// TIA Portal V19 export
FUNCTION_BLOCK "TYPIC_C104_IF_NSA"   // FB92, FBD
TITLE = TYPIC_C104_IF_NSA: Noodstroomaggregaat
{ S7_Optimized_Access := 'TRUE' }
AUTHOR : OCOTECH
FAMILY : Typical
NAME : C104.702
// Logisch Object Besturing: C104.702
// 
// De interne functie Noodstroomaggregaat verzorgt de bewaking van een noodstroomaggregaat.
// stored: MemoryReserve 10, SetENOAutomatically false
   VAR_INPUT
      EXT_AUT { ExternalAccessible := 'False'; ExternalVisible := 'False'; ExternalWritable := 'False'} : Bool;   // Externe (hoofd) beveiliging (1 = OK)
      EXT_HW { ExternalAccessible := 'False'; ExternalVisible := 'False'; ExternalWritable := 'False'} : Bool;   // Sturings hardware (PLC) bewaking (1 = OK)
      IN_STO_NOK { ExternalAccessible := 'False'; ExternalVisible := 'False'; ExternalWritable := 'False'} : Bool;   // Storing aanwezig die niet observeerbaar tot gevolg heeft
      IN_STO_OK { ExternalAccessible := 'False'; ExternalVisible := 'False'; ExternalWritable := 'False'} : Bool;   // Storing aanwezig die observeerbaarheid niet beinvloed
      IN_ENE { ExternalAccessible := 'False'; ExternalVisible := 'False'; ExternalWritable := 'False'} : Real;   // Geleverde energie per aggregaat
      IN_PHI { ExternalAccessible := 'False'; ExternalVisible := 'False'; ExternalWritable := 'False'} : Real;   // Fasehoek (cos phi)
      IN_SPA1 { ExternalAccessible := 'False'; ExternalVisible := 'False'; ExternalWritable := 'False'} : Real;   // Spanningsniveau lijn 1
      IN_SPA2 { ExternalAccessible := 'False'; ExternalVisible := 'False'; ExternalWritable := 'False'} : Real;   // Spanningsniveau lijn 2
      IN_SPA3 { ExternalAccessible := 'False'; ExternalVisible := 'False'; ExternalWritable := 'False'} : Real;   // Spanningsniveau lijn 3
      IN_STR { ExternalAccessible := 'False'; ExternalVisible := 'False'; ExternalWritable := 'False'} : Real;   // Stroomsterkte
      IN_WRE { ExternalAccessible := 'False'; ExternalVisible := 'False'; ExternalWritable := 'False'} : Bool;   // TRUE = werkingsregime: Belast FALSE = werkingsregime: Onbelast
      IN_STS1 { ExternalAccessible := 'False'; ExternalVisible := 'False'; ExternalWritable := 'False'} : Bool;   // Status: Standby
      IN_STS2 { ExternalAccessible := 'False'; ExternalVisible := 'False'; ExternalWritable := 'False'} : Bool;   // Status: Storing
      IN_STS3 { ExternalAccessible := 'False'; ExternalVisible := 'False'; ExternalWritable := 'False'} : Bool;   // Status: Uitgeschakeld
      IN_STS4 { ExternalAccessible := 'False'; ExternalVisible := 'False'; ExternalWritable := 'False'} : Bool;   // Status: Test
      IN_STS_AAN { ExternalAccessible := 'False'; ExternalVisible := 'False'; ExternalWritable := 'False'} : Bool;   // In bedrijf (Aan)
      IN_LDE { ExternalAccessible := 'False'; ExternalVisible := 'False'; ExternalWritable := 'False'} : Bool;   // Lekdetectie NSA
      IN_TYD_TOT_AAN_UUR { ExternalAccessible := 'False'; ExternalVisible := 'False'; ExternalWritable := 'False'} : LInt;   // TYD_TOT_AAN_UUR
      IN_SNS { ExternalAccessible := 'False'; ExternalVisible := 'False'; ExternalWritable := 'False'} : Bool;   // Noodstop (1 = gedeactiveerd)
      IN_OPT_LDE { ExternalAccessible := 'False'; ExternalVisible := 'False'; ExternalWritable := 'False'} : Bool;   // Lekdetectie brandstof dagtank
      IN_OPT_NIV { ExternalAccessible := 'False'; ExternalVisible := 'False'; ExternalWritable := 'False'} : Real;   // Brandstof niveau brandstof dagtank
      IN_OPT_HOOG { ExternalAccessible := 'False'; ExternalVisible := 'False'; ExternalWritable := 'False'} : Bool;   // Overvulbeveiliging brandstof dagtank aangesproken
      IN_OPT_STO { ExternalAccessible := 'False'; ExternalVisible := 'False'; ExternalWritable := 'False'} : Bool;   // Dagtank noodstroomaggregaat in storing
      IN_AUT_C104 { ExternalAccessible := 'False'; ExternalVisible := 'False'; ExternalWritable := 'False'} : Bool;   // Beveiligingen: serie geschakelde terugmelding (1 = OK)
   END_VAR
   VAR_OUTPUT
      VAR_IF_NSA { ExternalAccessible := 'False'; ExternalVisible := 'False'; ExternalWritable := 'False'} : "C104_VAR_IF_NSA_TYPIC";   // Struct met alle variabelen naar bovenliggende functies
   END_VAR
   VAR
      STO { ExternalWritable := 'False'} : Struct   // Storingen
         A001 : Bool;   // Beveiliging aangesproken
         A002 : Bool;   // Noodstroomaggregaat in storing
         A003 : Bool;   // Algemene storing noodstroomaggregaat
         A004 : Bool;   // Lekdetectie NSA
         A005 : Bool;   // Noodstop van het noodstroomaggregaat is geactiveerd
         A006 : Bool;   // Dagtank noodstroomaggregaat in storing
         A007 : Bool;   // Lekdetectie brandstof dagtank
         A008 : Bool;   // Overvulbeveiliging brandstof dagtank aangesproken
      END_STRUCT;
      VAR { ExternalWritable := 'False'} : Struct   // Variabelen
         ENE { ExternalAccessible := 'False'; ExternalVisible := 'False'} : Real;   // Geleverde energie per aggregaat [kWh]
         PHI { ExternalAccessible := 'False'; ExternalVisible := 'False'} : Real;   // Fasehoek (cos phi)
         SPA1 { ExternalAccessible := 'False'; ExternalVisible := 'False'} : Real;   // Spanningsniveau lijn 1
         SPA2 { ExternalAccessible := 'False'; ExternalVisible := 'False'} : Real;   // Spanningsniveau lijn 2
         SPA3 { ExternalAccessible := 'False'; ExternalVisible := 'False'} : Real;   // Spanningsniveau lijn 3
         STR { ExternalAccessible := 'False'; ExternalVisible := 'False'} : Real;   // Stroomsterkte
         WRE { ExternalAccessible := 'False'; ExternalVisible := 'False'} : Bool;   // TRUE = werkingsregime: Belast FALSE = werkingsregime: Onbelast
         STS1 { ExternalAccessible := 'False'; ExternalVisible := 'False'} : Bool;   // Status: Standby
         STS2 { ExternalAccessible := 'False'; ExternalVisible := 'False'} : Bool;   // Status: Storing
         STS3 { ExternalAccessible := 'False'; ExternalVisible := 'False'} : Bool;   // Status: Uitgeschakeld
         STS4 { ExternalAccessible := 'False'; ExternalVisible := 'False'} : Bool;   // Status: Test
         STS_AAN { ExternalAccessible := 'False'; ExternalVisible := 'False'} : Bool;   // In bedrijf (AAN)
         LDE { ExternalAccessible := 'False'; ExternalVisible := 'False'} : Bool;   // Lekdetectie NSA
         TYD_TOT_AAN_UUR { ExternalAccessible := 'False'; ExternalVisible := 'False'} : LInt;   // TYD_TOT_AAN_UUR
         SNS { ExternalAccessible := 'False'; ExternalVisible := 'False'} : Bool;   // Noodstop (1 = gedeactiveerd)
         OPT_LDE { ExternalAccessible := 'False'; ExternalVisible := 'False'} : Bool;   // Lekdetectie brandstof dagtank
         OPT_NIV { ExternalAccessible := 'False'; ExternalVisible := 'False'} : Real;   // Brandstof niveau brandstof dagtank
         OPT_HOOG { ExternalAccessible := 'False'; ExternalVisible := 'False'} : Bool;   // Overvulbeveiliging brandstof dagtank aangesproken
         OPT_STO { ExternalAccessible := 'False'; ExternalVisible := 'False'} : Bool;   // Dagtank noodstroomaggregaat in storing
         EXT_AUT { ExternalAccessible := 'False'; ExternalVisible := 'False'} : Bool;   // Externe (hoofd) beveiliging aangesproken
         EXT_HW { ExternalAccessible := 'False'; ExternalVisible := 'False'} : Bool;   // Sturings hardware (PLC) in storing
      END_STRUCT;
   END_VAR
BEGIN

REGION Network 1: START
END_REGION

REGION Network 2: +++ Verwerking meetwaarden en statussen +++
   // De meetwaarden en statussen van het noodstroomaggregaat worden ontvangen vanuit de interne sturing.
END_REGION

REGION Network 3: +++ Storingen +++
   // Verwerken van de storingsmeldingen (inputs).
END_REGION

REGION Network 4: Storing A001: Beveiliging aangesproken
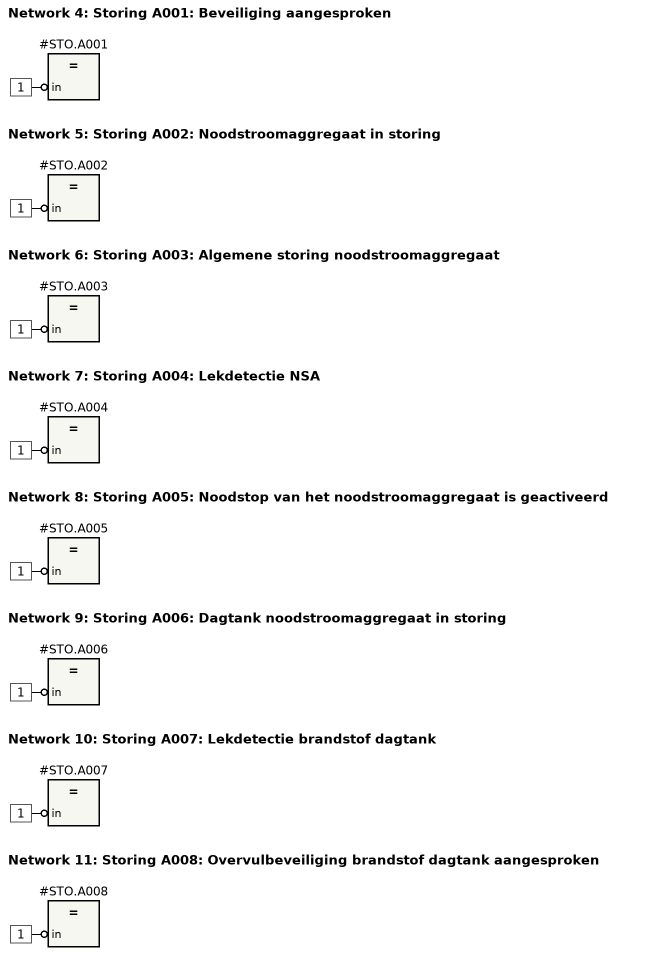
   #STO.A001 := NOT 1;
END_REGION

REGION Network 5: Storing A002: Noodstroomaggregaat in storing
   #STO.A002 := NOT 1;
END_REGION

REGION Network 6: Storing A003: Algemene storing noodstroomaggregaat
   #STO.A003 := NOT 1;
END_REGION

REGION Network 7: Storing A004: Lekdetectie NSA
   #STO.A004 := NOT 1;
END_REGION

REGION Network 8: Storing A005: Noodstop van het noodstroomaggregaat is geactiveerd
   #STO.A005 := NOT 1;
END_REGION

REGION Network 9: Storing A006: Dagtank noodstroomaggregaat in storing
   #STO.A006 := NOT 1;
END_REGION

REGION Network 10: Storing A007: Lekdetectie brandstof dagtank
   #STO.A007 := NOT 1;
END_REGION

REGION Network 11: Storing A008: Overvulbeveiliging brandstof dagtank aangesproken
   #STO.A008 := NOT 1;
END_REGION

REGION Network 12 (SCL): EINDE
   // Variabelen van intern scada rakvlak naar outputs copieren
   #VAR_IF_NSA.ENE := #VAR.ENE;
   #VAR_IF_NSA.PHI := #VAR.PHI;
   #VAR_IF_NSA.SPA1 := #VAR.SPA1;
   #VAR_IF_NSA.SPA2 := #VAR.SPA2;
   #VAR_IF_NSA.SPA3 := #VAR.SPA3;
   #VAR_IF_NSA.STR := #VAR.STR;
   #VAR_IF_NSA.WRE := #VAR.WRE;
   #VAR_IF_NSA.STS1 := #VAR.STS1;
   #VAR_IF_NSA.STS2 := #VAR.STS2;
   #VAR_IF_NSA.STS3 := #VAR.STS3;
   #VAR_IF_NSA.STS4 := #VAR.STS4;
   #VAR_IF_NSA.STS_AAN := #VAR.STS_AAN;
   #VAR_IF_NSA.LDE := #VAR.LDE;
   #VAR_IF_NSA.TYD_TOT_AAN_UUR := #VAR.TYD_TOT_AAN_UUR;
   #VAR_IF_NSA.SNS := #VAR.SNS;
   #VAR_IF_NSA.OPT_LDE := #VAR.OPT_LDE;
   #VAR_IF_NSA.OPT_NIV := #VAR.OPT_NIV;
   #VAR_IF_NSA.OPT_HOOG := #VAR.OPT_HOOG;
   #VAR_IF_NSA.OPT_STO := #VAR.OPT_STO;
   #VAR_IF_NSA.EXT_AUT := #VAR.EXT_AUT;
   #VAR_IF_NSA.EXT_HW := #VAR.EXT_HW;
   #VAR_IF_NSA.STO := #STO;
END_REGION
END_FUNCTION_BLOCK
